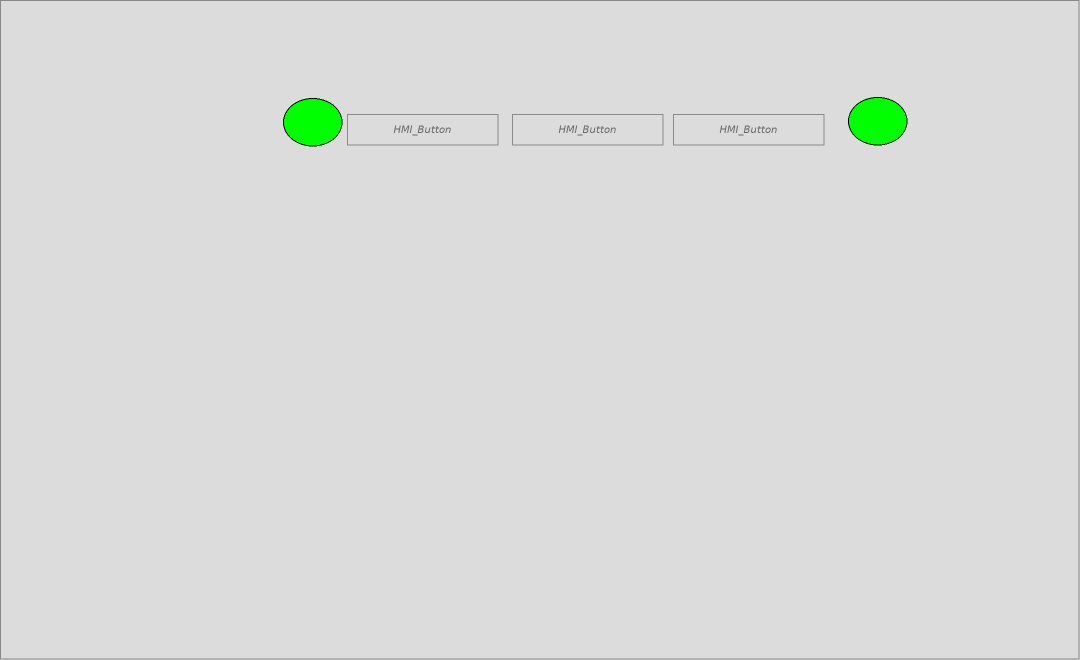
VISUALIZATION Page_Infeed  // 1080x660, background image 
    Frame (347,114 151x31)
        shows HMI_Button(i_sText := 'Open', iq_stButton := GVL_Modules.g_emInfeedConveyor.s_cmDoor.s_stHmi.btnOpenDoor.s_stHmi)
    Frame (673,114 151x31)
        shows HMI_Button(i_sText := 'Close', iq_stButton := GVL_Modules.g_emInfeedConveyor.s_cmDoor.s_stHmi.btnCloseDoor.s_stHmi)
    Frame (512,114 151x31)
        shows HMI_Button(i_sText := 'Stop', iq_stButton := GVL_Modules.g_emInfeedConveyor.s_cmDoor.s_stHmi.btnStopDoor.s_stHmi)
    Ellipse (283,98 59x48), colour toggle: not GVL_Modules.g_emInfeedConveyor.s_cmDoor.s_stHmi.bStaDoorOpen
    Ellipse (848,97 59x48), colour toggle: not GVL_Modules.g_emInfeedConveyor.s_cmDoor.s_stHmi.bStaDoorCLosed
END_VISUALIZATION

(* stored: Version 1.1.0.1
   Visu Page_Infeed: Id {fa9497d4-317f-4852-864b-de4603a02a9c} *)
